FUNCTION_BLOCK X2Y2_FBD (* Compute X^2-Y^2 in FBD *)
  (* Standard: 61499-1 *)
  (* Version 0.0, 2003-08-11, JHC, Rockwell Automation, Derived from FB_X2Y2_ST. *)
  (* Compiler header: package fb.rt.student; import fb.rt.plc.math.*; *)
  (* Compiler Java IBM Jikes 1.0.6 *)
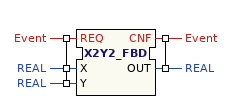
  EVENT_INPUT
    REQ WITH X, Y;
  END_EVENT
  EVENT_OUTPUT
    CNF WITH OUT;
  END_EVENT
  VAR_INPUT
    X : REAL;
    Y : REAL;
  END_VAR
  VAR_OUTPUT
    OUT : REAL;
  END_VAR
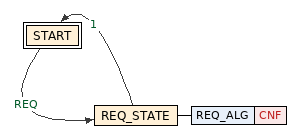
  EC_STATES
    START;
    REQ_STATE : REQ_ALG -> CNF;
  END_STATES
  EC_TRANSITIONS
    START TO REQ_STATE := REQ;
    REQ_STATE TO START := 1;
  END_TRANSITIONS
  ALGORITHM REQ_ALG IN FBD:
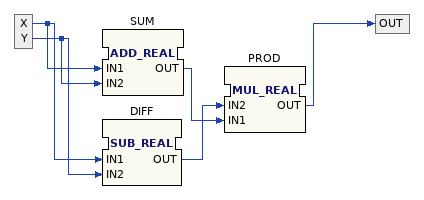
    FBS
      SUM : ADD_REAL;
      DIFF : SUB_REAL;
      PROD : MUL_REAL;
    END_FBS
    DATA_CONNECTIONS
      X TO SUM.IN1;
      X TO DIFF.IN1;
      Y TO SUM.IN2;
      Y TO DIFF.IN2;
      DIFF.OUT TO PROD.IN2;
      SUM.OUT TO PROD.IN1;
      PROD.OUT TO OUT;
    END_CONNECTIONS
  END_ALGORITHM
END_FUNCTION_BLOCK
